// SIMATIC STEP 7 (V5.x) project PROBLEM 4
// CPU: CPU 314C-2 DP
// station: Hardware
// station: SIMATIC 300(1)
// station: P_ADR_BUS
// program: S7 Program(1)

ORGANIZATION_BLOCK OB 1
TITLE = "Main Program Sweep (Cycle)"
//Problem 4
VERSION : 0.1
VAR_TEMP
  OB1_EV_CLASS : BYTE ;	//Bits 0-3 = 1 (Coming event), Bits 4-7 = 1 (Event class 1)
  OB1_SCAN_1 : BYTE ;	//1 (Cold restart scan 1 of OB 1), 3 (Scan 2-n of OB 1)
  OB1_PRIORITY : BYTE ;	//Priority of OB Execution
  OB1_OB_NUMBR : BYTE ;	//1 (Organization block 1, OB1)
  OB1_RESERVED_1 : BYTE ;	//Reserved for system
  OB1_RESERVED_2 : BYTE ;	//Reserved for system
  OB1_PREV_CYCLE : INT ;	//Cycle time of previous OB1 scan (milliseconds)
  OB1_MIN_CYCLE : INT ;	//Minimum cycle time of OB1 (milliseconds)
  OB1_MAX_CYCLE : INT ;	//Maximum cycle time of OB1 (milliseconds)
  OB1_DATE_TIME : DATE_AND_TIME ;	//Date and time OB1 started
END_VAR
BEGIN
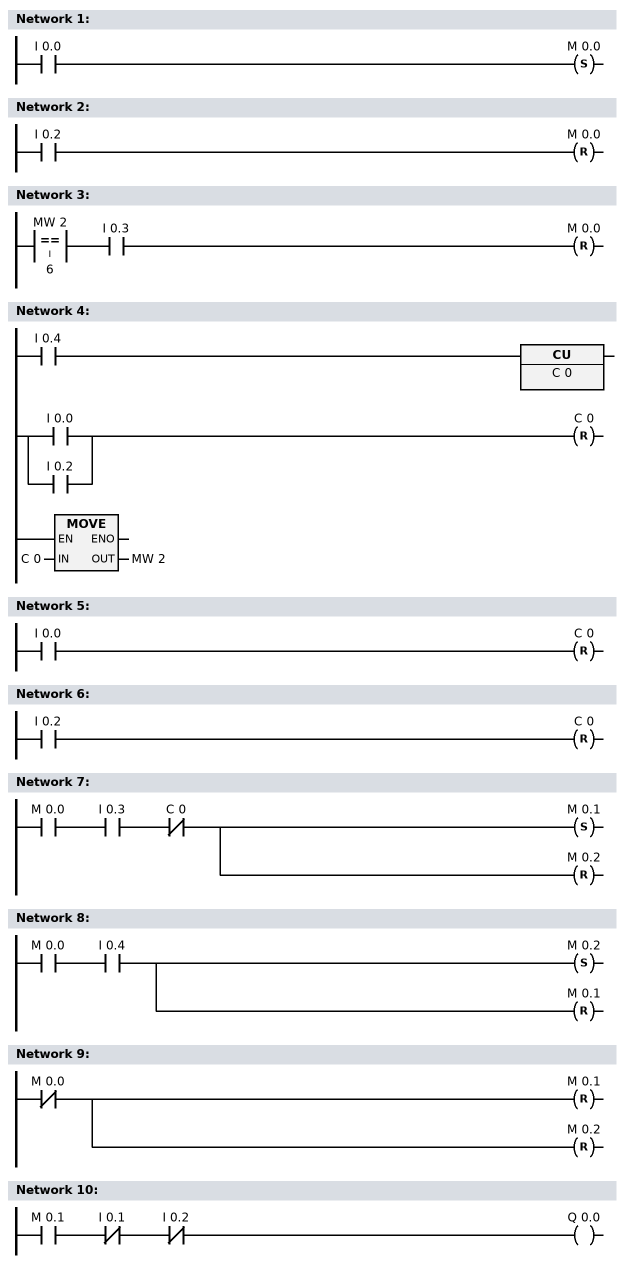
NETWORK
TITLE =
      A     I 0.0;
      S     M 0.0;
NETWORK
TITLE =
      A     I 0.2;
      R     M 0.0;
NETWORK
TITLE =
      A(;
      L     MW 2;
      L     6;
      ==I;
      );
      A     I 0.3;
      R     M 0.0;
NETWORK
TITLE =
      A     I 0.4;
      CU    C 0;
      BLD   101;
      NOP   0;
      NOP   0;
      A(;
      O     I 0.0;
      O     I 0.2;
      );
      R     C 0;
      L     C 0;
      T     MW 2;
      NOP   0;
      NOP   0;
NETWORK
TITLE =
      A     I 0.0;
      R     C 0;
NETWORK
TITLE =
      A     I 0.2;
      R     C 0;
NETWORK
TITLE =
      A     M 0.0;
      A     I 0.3;
      AN    C 0;
      S     M 0.1;
      R     M 0.2;
NETWORK
TITLE =
      A     M 0.0;
      A     I 0.4;
      S     M 0.2;
      R     M 0.1;
NETWORK
TITLE =
      AN    M 0.0;
      R     M 0.1;
      R     M 0.2;
NETWORK
TITLE =
      A     M 0.1;
      AN    I 0.1;
      AN    I 0.2;
      =     Q 0.0;
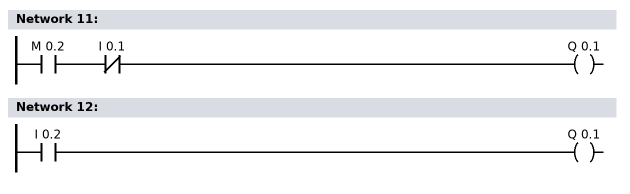
NETWORK
TITLE =
      A     M 0.2;
      AN    I 0.1;
      =     Q 0.1;
NETWORK
TITLE =
      A     I 0.2;
      =     Q 0.1;
END_ORGANIZATION_BLOCK
